Fanuc KAREL source: CA0115.KL

-- PROVISIONAL review KL for V770-1; original PC SHA256 acf8a7bfe4bd941e6ff2baed8ec0bb468f60d2fe39a1568b635cdf1c82b04070
-- Incomplete behavior may be omitted. Consult companion uncertainty JSON. Do not deploy.
PROGRAM CA0115
%NOLOCKGROUP
BEGIN
  -- UNRESOLVED_PC offsets 0-1; opcodes 7B
  -- UNRESOLVED_PC offsets 6-16; opcodes 2D,7F
  -- UNRESOLVED_PC offsets 21-25; opcodes 7F
  -- UNRESOLVED_PC offsets 30-37; opcodes 9C,23
  -- UNRESOLVED_PC offsets 42-49; opcodes 9D,23
  -- UNRESOLVED_PC offsets 54-65; opcodes 2E,23
  -- UNRESOLVED_PC offsets 70-77; opcodes 9D,23
  -- UNRESOLVED_PC offsets 82-91; opcodes 3F,75
  -- UNRESOLVED_PC offsets 96-110; opcodes 2E,22,9D,33,35
  -- UNRESOLVED_PC offsets 115-129; opcodes 2E,22,9D,33,35
  -- UNRESOLVED_PC offsets 134-149; opcodes 2E,22,32,35
  -- UNRESOLVED_PC offsets 154-169; opcodes 2E,22,32,35
  -- UNRESOLVED_PC offsets 174-280; opcodes 27,22,22,22,22,22,22,22,22,22,22,22,22,22,22,22,22,AA,23
  -- UNRESOLVED_PC offsets 285-289; opcodes 7F
END CA0115
